{attribute 'call_after_init'}
FUNCTION_BLOCK TcpDataQueue
VAR
	elements : FB_BA_DynamicArray := (uiEntrySize := SIZEOF(POINTER TO TcpData), uiMinExpCount := GVL.initArraySize); 
	length : INT := 0;
	
	entrySize : UDINT;
END_VAR
(*
this container stores dynamically generated AdsData Structs
AdsData to be added are passed by reference, then this function block allocates a structure to be stored
AdsData are get() by reference and poll() by value
*)

METHOD clear : BOOL
VAR
	i : INT;
	temp : REFERENCE TO TcpData;
	tempAdr : POINTER TO TcpData;
END_VAR
FOR i:=0 TO length-1 BY 1 DO
	temp := get(index := i, getSize => );
	tempAdr := ADR(temp);
	__DELETE(tempAdr);
END_FOR

elements.Reset();
length := 0;
END_METHOD

METHOD contains : BOOL //check contents, not pointer value
VAR_INPUT
	value : REFERENCE TO TcpData;
END_VAR
VAR_OUTPUT
	atIndex : INT;
END_VAR
VAR
	temp : REFERENCE TO TcpData;
	i : INT;
END_VAR
IF length = 0 THEN
	contains := FALSE;
	RETURN;
END_IF

FOR i:=0 TO length-1 BY 1 DO
	temp := get(index := i, getSize => );
	
	IF 
		SIZEOF(value) = entrySize AND //same size
		MEMCMP(ADR(temp), ADR(value), SIZEOF(entrySize)) = 0 //same data
	THEN
		contains := TRUE;
		atIndex := i;
		RETURN;
	END_IF
	
END_FOR
contains := FALSE;
END_METHOD

METHOD get : REFERENCE TO TcpData
VAR_INPUT
	index : INT;
END_VAR
VAR_OUTPUT
	getSize : UDINT;
END_VAR
IF length = 0 OR index < 0 OR index >= length THEN
	getSize := 0;
ELSE
	elements.GetEntry(diIndex := index, pResultEntry := ADR(get));
	getSize := SIZEOF(get);
END_IF
END_METHOD

METHOD isEmpty : BOOL
VAR_INPUT
END_VAR
isEmpty := length = 0;
END_METHOD

METHOD poll : TcpData
VAR_OUTPUT
	getSize : UDINT;
END_VAR
IF length > 0 THEN
	poll := get(index := 0, getSize => getSize);
	elements.RemoveEntry(diIndex := 0);
	
	length := length - 1;
END_IF
END_METHOD

METHOD push : BOOL
VAR_INPUT
	value : REFERENCE TO TcpData;
END_VAR
VAR
	temp : POINTER TO TcpData;
END_VAR
temp := __NEW(TcpData);
temp^ := value;

elements.AddEntryPtr(pEntry := temp);

length := length + 1;
END_METHOD

METHOD set : BOOL
VAR_INPUT
	i : INT;
	value : REFERENCE TO TcpData;
END_VAR
VAR
	temp : REFERENCE TO TcpData;
END_VAR
IF length = 0 THEN
	RETURN;
END_IF

IF i >= 0 AND i < length THEN
	temp REF= get(i);
	temp := value;
	
	set := TRUE;
END_IF
END_METHOD

{attribute 'call_after_init'}
METHOD setup : BOOL
VAR_INPUT
END_VAR
entrySize := SIZEOF(TcpData);
END_METHOD

METHOD size : INT
size := length;
END_METHOD

END_FUNCTION_BLOCK

(* stored: Version 1.1.0.1, ProductVersion 3.1.4024.11
   POU TcpDataQueue: Id {31746788-719c-4a8b-a524-0166dcbe980e}, SpecialFunc None
   Method clear: Id {7e6b7cd5-5398-4417-b26e-22e0dbcb02e8}
   Method contains: Id {07e710ce-08fc-4292-bc18-49f03592976a}
   Method get: Id {9e57ab30-80ce-4738-b192-a7e941806aa3}
   Method isEmpty: Id {da97b880-8db9-4424-8843-9ec29b6037f1}
   Method poll: Id {961519c6-422e-4129-9154-3b267d33e6ec}
   Method push: Id {c4f1a3cb-e929-4827-a82b-2256280acdc8}
   Method set: Id {1e3569ba-9059-42e0-9fbd-dade77d8a158}
   Method setup: Id {b542d38b-f2d6-4cb2-a697-0dd1c38090ad}
   Method size: Id {00d5a93a-5526-4eb3-be4a-cc3cac69328d} *)
